FUNCTION F_CubitCalculate : lreal
VAR_INPUT
	A : LREAL;
	B : LREAL;
	C : LREAL;
	D : LREAL;
	x : LREAL;
END_VAR
VAR_OUTPUT
	Y : LREAL;
END_VAR

Y := A*x*x*x + B*x*x + C*x + D;
F_CubitCalculate := Y;

END_FUNCTION

(* stored: Version 1.1.0.1, ProductVersion 3.1.4024.12
   POU F_CubitCalculate: Id {b1c0162c-5c4b-45b0-a476-ed5b15f8ca38}, SpecialFunc None *)
